// TIA Portal V19 export
DATA_BLOCK "DI_FW_HUB_rechts"   // DB23
AUTHOR : MS
// stored: AutoNumber false, InstanceOfName FB_HUB_FW_re, InstanceOfType FB
"FB_HUB_FW_re"
   // VAR_INPUT
   //    FW_DBNr : Int;
   //    SysTime : Time;
   // END_VAR
   // VAR RETAIN
   //    Config : Struct
   //       Speed : Struct
   //          Min : Int;
   //          Tipp : Int;
   //          Hand : Int;
   //          Max : Int;
   //          Norm : Real;
   //          endMess : Real;
   //       END_STRUCT;
   //       Rampe : Struct
   //          Auf_Heben : Real;
   //          Ab_Heben : Real;
   //          Auf_Senken : Real;
   //          Ab_Senken : Real;
   //          NotStop : Real;
   //       END_STRUCT;
   //       Bereich : Struct
   //          Pos : DInt;
   //          Stop : DInt;
   //          Ziel : DInt;
   //          Absetzen : DInt;
   //          Langsam : DInt;
   //       END_STRUCT;
   //       TV_Position : DInt;
   //       Reaktionszeit : Int;
   //       Startzeit : Int;
   //       Variante : Byte;
   //       SimIstSpeed : Byte;
   //       SimSensors : DWord;
   //       SimTakt : DInt;
   //    END_STRUCT;
   //    IN : Struct
   //       BA_Tipp : Bool;
   //       BA_Hand : Bool;
   //       BA_Auto : Bool;
   //       Heben_aktiv : Bool;
   //       Frg_Hub : Bool;
   //       Frg_Eil : Bool;
   //       Break_on : Bool;
   //       mittig : Bool;
   //       resB : Byte;
   //       HubInc : DInt;
   //       ZielInc : DInt;
   //       Absetz_Inc : DInt;
   //       IstSpeed : Int;
   //    END_STRUCT;
   //    OUT : Struct
   //       Hub_Ok : Bool;
   //       Break_off : Bool;
   //       res_1 : Bool;
   //       res_2 : Bool;
   //       res_3 : Bool;
   //       res_4 : Bool;
   //       res_5 : Bool;
   //       res_6 : Bool;
   //       resB : Byte;
   //       Bereich_langsam : DInt;
   //       SollSpeed : Int;
   //    END_STRUCT;
   //    Tmp : Struct
   //       lastTime : DInt;
   //       DiffTime : Real;
   //       lastSpeed : Real;
   //       Messung : Struct
   //          lastInc : Real;
   //          addInc : Real;
   //          addTime : Real;
   //          lastIst : Int;
   //          messAct : Bool;
   //       END_STRUCT;
   //       StopCount : DInt;
   //       subInc : Real;
   //       lastOut : Real;
   //       TaktCount : Real;
   //       PtrSensors : DWord;
   //       RunTime : DInt;
   //    END_STRUCT;
   // END_VAR
BEGIN
END_DATA_BLOCK
